FUNCTION_BLOCK FB_DistanceSensor IMPLEMENTS ITF_SubSystem
VAR_OUTPUT
	fDistance 			: LREAL;
END_VAR
VAR
	//Local
	fbEL6021			: FB_SerialComRS422;

	//ErrorBits
	bCommunicationError : BIT;
	bOutOfRange 		: BIT;
END_VAR
VAR CONSTANT
	fSMR 		: LREAL := 50.0;				// Start of Measuring Range
	fEMR 		: LREAL := 150.0;				// End of Measuring Range
END_VAR

fbEL6021(stReceiveData:=DistanceSensor.stEL6021In, stTransmitData:=DistanceSensor.stEL6021Out);

fDistance := fbEL6021.fDistance;

METHOD PRIVATE doCheckRange : BOOL
VAR_INPUT
	fDistanceValue : LREAL;
	fMax : LREAL;
	fMin : LREAL;
END_VAR
IF fDistanceValue < fMin OR fDistanceValue > fMax THEN
	doCheckRange := FALSE;
ELSE
	doCheckRange := TRUE;
END_IF
END_METHOD

PROPERTY eCondition : SubLevelCondition
GET
IF nErrorID <> 0 THEN
	eCondition := SubLevelCondition.ERROR;
ELSE
	eCondition := SubLevelCondition.RUN;
END_IF
END_GET
END_PROPERTY

PROPERTY nErrorID : UDINT
GET
IF fbEL6021.eReceiveErrorID <> COMERROR_NOERROR THEN
	bCommunicationError := TRUE;
ELSE
	bCommunicationError := FALSE;
END_IF

bOutOfRange := NOT doCheckRange(fDistanceValue:= fDistance, fMax:=fEMR, fMin:=fSMR);

nErrorID.0 := bCommunicationError;
nErrorID.1 := bOutOfRange;
END_GET
END_PROPERTY

END_FUNCTION_BLOCK

(* stored: Version 1.1.0.1, ProductVersion 3.1.4024.12
   POU FB_DistanceSensor: Id {f4605cef-c88d-437c-8e3e-a6c190169adb}, SpecialFunc None
   Method doCheckRange: Id {f0fc130c-4d4c-401a-8605-074ef0591044}
   Property eCondition: Id {dec3797b-3659-4283-97b1-3349172eac00}
   Get Get: Id {a432a058-d6e8-46c9-ab20-17a501839623}
   Property nErrorID: Id {802f66c6-09e3-4b76-b004-cc262d9b1836}
   Get Get: Id {afc3c74c-8e96-49c4-b480-aa4a6067a1e9} *)
